FUNCTION F_ITC_SendTTC : BOOL
(**************************************************************************************
 * 	Application		:	BoxControl Framework
 *	Revision		:	$Revision: 404529 $
 *	Revision date	:	$Date: 2018-04-23 08:21:38 +0200 (Mo., 23 Apr 2018) $
 *	Last changed by	:	$Author: b7bolm $
 *	URL				:	$URL: http://almscdc.swisslog.com/repo/SWPD/Development/BoxControlFramework/20_Release/trunk/01_Software/BCF/BCF/JumpStart/20_Product/10_App/11_Com/10_Lib/10_Conv/11_ITC/F_ITC_SendTTC.TcPOU $
 *
 *	Purpose			:	Wrap message - TTC
 *
 * ------------------------------------------------------------------------------------
 *	Copyright Swisslog [IP AG], Switzerland. All rights reserved.
 * 
 * ------------------------------------------------------------------------------------
 *	
 * 	Revision History: 
 *
 * 	VERSION			DATE			INITIALS			DESCRIPTION
 *	0.1				01.01.2001		swl					Example
 *
 **************************************************************************************)
VAR_INPUT
	eChannelSrc		: E_MFCS_Channel; // Source communicaton channel		
	PositionName	: STRING(Conveyor.POSITION_STRINGLENGTH); // Position
	TU_DataIndex	: DINT; // TU-DataIndex
	MsgSequence		: INT; // Assignment message sequence
	TU_ID			: STRING(Conveyor.TU_ID_STRINGLENGTH); // 18 Digit SSID
	AssignmentID	: UDINT; // assignment id
	eReturnCode		: E_ErrorConv; // Return code
END_VAR
VAR
	TTC				: ST_ITC_TTC; 
END_VAR

// Map values
TTC.Position := PositionName;
TTC.TU_DataIndex := TU_DataIndex;
TTC.MsgSequence := MsgSequence;
TTC.TU_ID := TU_ID;
TTC.AssignmentID := AssignmentID;
TTC.ReturnCode := eReturnCode;

// Forward to ITC
F_ITC_SendTTC := fbITC_Manager.M_SendData(
					meChannel	:= eChannelSrc,
					mMsgType	:= E_ITC_MsgTypeConv.TRANSPORT_TASK_COMPLETE,
					mpData		:= ADR(TTC),
					mLen		:= SIZEOF(TTC));

END_FUNCTION

(* stored: Version 1.1.0.1, ProductVersion 3.1.4022.12
   POU F_ITC_SendTTC: Id {96c6a951-4768-4823-96ba-4b2973ecbb31}, SpecialFunc None *)
